TYPE E_ServStates :
(**************************************************************************************
 * 	AUTHOR		Swisslog
 * 	LIBRARY		Data types/02_Library/02_Communication/TCP-Driver
 *	RELEASE		1.0.0
 * ------------------------------------------------------------------------------------
 * 	Revision History: 
 *
 * 	VERSION		DATE		INITIALS	DESCRIPTION
 *	0.1		07.09.2011	swl		initial version
 **************************************************************************************)
(
	ACCEPT_IDLE,
	ACCEPT_OPEN_START,
	ACCEPT_OPEN_WAIT,
	CLIENT_CONNECTED,
	ACCEPT_CLOSE_START,
	ACCEPT_CLOSE_WAIT,
	ACCEPT_ERROR
);
END_TYPE

(* stored: Version 1.1.0.1, ProductVersion 3.1.4020.6
   DUT E_ServStates: Id {f2c8f2e8-dcb6-4baa-a1b9-08be82f281f1} *)
